(* IEC 61131-3 sources: stc/tests/type_system, 4 files *)

(* ---- init_test.st ---- *)
(* Initialiser test suite (RUNT-06)
   Array, repetition, struct-array, TYPE default and FB-instance
   initialisers apply when the variable is instantiated. Literals are typed
   where the checker's literal adoption would otherwise matter.
*)

TYPE ST_Item :
STRUCT
    id : INT := INT#5;
    name : STRING := 'x';
END_STRUCT
END_TYPE

TYPE T_Speed : INT := INT#50; END_TYPE

FUNCTION_BLOCK FB_Base
VAR
    base_x : INT := INT#3;
END_VAR
END_FUNCTION_BLOCK

FUNCTION_BLOCK FB_Drive EXTENDS FB_Base
VAR_INPUT
    speed : INT;
END_VAR
VAR
    tbl : ARRAY[1..2] OF INT := [INT#4, INT#5];
    item : ST_Item := (name := 'drive');
END_VAR
END_FUNCTION_BLOCK

VAR_GLOBAL CONSTANT
    N_ITEMS : INT := 3;
END_VAR

TEST_CASE 'Array initialiser'
VAR
    arr : ARRAY[1..3] OF INT := [INT#1, INT#2, INT#3];
END_VAR
    ASSERT_EQ(arr[1], INT#1);
    ASSERT_EQ(arr[2], INT#2);
    ASSERT_EQ(arr[3], INT#3);
END_TEST_CASE

TEST_CASE 'Repetition and tail defaults'
VAR
    rep : ARRAY[1..5] OF INT := [3(INT#0), INT#7];
END_VAR
    ASSERT_EQ(rep[3], INT#0);
    ASSERT_EQ(rep[4], INT#7);
    ASSERT_EQ(rep[5], INT#0);
END_TEST_CASE

TEST_CASE 'Struct array over a GVL constant bound'
VAR
    items : ARRAY[1..init_test.N_ITEMS] OF ST_Item := [(id := INT#1, name := 'a'), (id := INT#2)];
END_VAR
    ASSERT_EQ(items[1].name, 'a');
    ASSERT_EQ(items[2].id, INT#2);
    ASSERT_EQ(items[2].name, 'x');
    ASSERT_EQ(items[3].id, INT#5);
END_TEST_CASE

TEST_CASE 'TYPE defaults'
VAR
    s : ST_Item;
    v : T_Speed;
END_VAR
    ASSERT_EQ(s.id, INT#5);
    ASSERT_EQ(v, INT#50);
END_TEST_CASE

TEST_CASE 'FB instances get their own initialised members'
VAR
    d1 : FB_Drive;
    d2 : FB_Drive := (speed := INT#9);
END_VAR
    ASSERT_EQ(d1.base_x, INT#3);
    ASSERT_EQ(d2.tbl[2], INT#5);
    ASSERT_EQ(d2.speed, INT#9);
    d1.item.name := 'changed';
    ASSERT_EQ(d2.item.name, 'drive');
END_TEST_CASE

(* ---- all_types.st ---- *)
(* All Types Declaration File
   Exercises every IEC 61131-3 type supported by the stc toolchain:
   elementary types, arrays, structs, enums, subranges, strings.
*)

(* Enum type declaration *)
TYPE MachineState : (
    MS_IDLE := 0,
    MS_RUNNING := 1,
    MS_FAULT := 2,
    MS_MAINTENANCE := 3
);
END_TYPE

(* Struct type declaration *)
TYPE SensorReading :
STRUCT
    Value     : REAL;
    RawCount  : INT;
    Valid     : BOOL;
    Timestamp : DINT;
    TagName   : STRING;
END_STRUCT;
END_TYPE

(* Subrange type *)
TYPE PercentRange : INT (0..100);
END_TYPE

TYPE MotorSpeed : REAL (0.0..1500.0);
END_TYPE

(* Program using all types *)
PROGRAM TypeShowcase
VAR
    (* Boolean *)
    bFlag : BOOL := TRUE;
    bLatch : BOOL := FALSE;

    (* Integer types *)
    nSint : SINT := -10;
    nInt  : INT := 1000;
    nDint : DINT := 100000;
    nLint : LINT := 1000000;

    (* Unsigned integer types *)
    nUsint : USINT := 200;
    nUint  : UINT := 50000;
    nUdint : UDINT := 4000000;
    nUlint : ULINT := 8000000;

    (* Bit string types *)
    bByte  : BYTE := 16#FF;
    wWord  : WORD := 16#ABCD;
    dwDword : DWORD := 16#12345678;
    lwLword : LWORD := 16#FEDCBA98;

    (* Real types *)
    fReal  : REAL := 3.14;
    fLreal : LREAL := 2.718281828;

    (* String types *)
    sName  : STRING := 'Hello World';
    sEmpty : STRING := '';

    (* Time types *)
    tDelay : TIME := T#500ms;
    tCycle : TIME := T#100ms;

    (* Array *)
    aTemps : ARRAY[1..10] OF REAL;
    aFlags : ARRAY[0..7] OF BOOL;

    (* Enum instance *)
    eState : MachineState := MS_IDLE;

    (* Struct instance *)
    stSensor : SensorReading;

    (* Loop variable *)
    i : INT;
END_VAR
    (* Exercise boolean operators *)
    bLatch := bFlag AND NOT bLatch;
    bLatch := bFlag OR bLatch;
    bLatch := bFlag XOR bLatch;

    (* Exercise integer arithmetic *)
    nInt := nInt + 1;
    nDint := nDint * 2;
    nLint := nLint - 500;

    (* Exercise real arithmetic *)
    fReal := fReal * 2.0;
    fLreal := fLreal + 1.0;

    (* Array operations *)
    FOR i := 1 TO 10 DO
        aTemps[i] := INT_TO_REAL(i) * 10.5;
    END_FOR;

    aFlags[0] := TRUE;
    aFlags[7] := FALSE;

    (* Enum usage *)
    eState := MS_RUNNING;
    IF eState = MS_RUNNING THEN
        nInt := nInt + 100;
    END_IF;

    (* Struct field access *)
    stSensor.Value := 25.4;
    stSensor.RawCount := 1023;
    stSensor.Valid := TRUE;
    stSensor.TagName := 'TT-101';

    (* String operations *)
    sName := CONCAT(sName, '!');
END_PROGRAM

(* ---- type_test.st ---- *)
(* Type System Test Suite
   Validates all elementary types, arithmetic, conversions,
   string operations, arrays, and control flow constructs.
*)

TEST_CASE 'Integer arithmetic on all widths'
VAR
    nSint : SINT := 10;
    nInt  : INT := 1000;
    nDint : DINT := 100000;
    nLint : LINT := 1000000;
END_VAR
    nSint := nSint + 5;
    ASSERT_EQ(nSint, 15);

    nInt := nInt * 2;
    ASSERT_EQ(nInt, 2000);

    nDint := nDint - 50000;
    ASSERT_EQ(nDint, 50000);

    nLint := nLint + 500000;
    ASSERT_EQ(nLint, 1500000);
END_TEST_CASE

TEST_CASE 'Unsigned integer types'
VAR
    nUsint : USINT := 200;
    nUint  : UINT := 50000;
    nUdint : UDINT := 4000000;
END_VAR
    nUsint := nUsint + 55;
    ASSERT_EQ(nUsint, 255);

    nUint := nUint - 10000;
    ASSERT_EQ(nUint, 40000);

    nUdint := nUdint * 2;
    ASSERT_EQ(nUdint, 8000000);
END_TEST_CASE

TEST_CASE 'REAL arithmetic and ASSERT_NEAR'
VAR
    fReal  : REAL := 3.14;
    fLreal : LREAL := 2.718281828;
    result : REAL;
END_VAR
    result := fReal * 2.0;
    ASSERT_NEAR(result, 6.28, 0.001);

    fLreal := fLreal + 1.0;
    ASSERT_NEAR(fLreal, 3.718281828, 0.000001);

    (* Division *)
    result := 10.0 / 3.0;
    ASSERT_NEAR(result, 3.333333, 0.001);
END_TEST_CASE

TEST_CASE 'Boolean logic operators'
VAR
    a : BOOL := TRUE;
    b : BOOL := FALSE;
    r : BOOL;
END_VAR
    r := a AND b;
    ASSERT_FALSE(r);

    r := a OR b;
    ASSERT_TRUE(r);

    r := a XOR b;
    ASSERT_TRUE(r);

    r := NOT a;
    ASSERT_FALSE(r);

    r := a AND NOT b;
    ASSERT_TRUE(r);

    (* Double negation *)
    r := NOT NOT a;
    ASSERT_TRUE(r);
END_TEST_CASE

TEST_CASE 'Comparison operators'
VAR
    x : INT := 10;
    y : INT := 20;
END_VAR
    ASSERT_TRUE(x < y);
    ASSERT_TRUE(y > x);
    ASSERT_TRUE(x <= 10);
    ASSERT_TRUE(y >= 20);
    ASSERT_TRUE(x <> y);
    ASSERT_FALSE(x = y);
    ASSERT_TRUE(x = 10);
END_TEST_CASE

TEST_CASE 'Type conversions INT to REAL'
VAR
    n : INT := 42;
    f : REAL;
END_VAR
    f := INT_TO_REAL(n);
    ASSERT_NEAR(f, 42.0, 0.01);
END_TEST_CASE

TEST_CASE 'Type conversions REAL to INT'
VAR
    f : REAL := 3.7;
    n : INT;
END_VAR
    n := REAL_TO_INT(f);
    ASSERT_EQ(n, 4);  (* Banker's rounding: 3.7 rounds to 4 *)
END_TEST_CASE

TEST_CASE 'Type conversions BOOL to INT and back'
VAR
    b : BOOL := TRUE;
    n : INT;
    b2 : BOOL;
END_VAR
    n := BOOL_TO_INT(b);
    ASSERT_EQ(n, 1);

    b2 := INT_TO_BOOL(0);
    ASSERT_FALSE(b2);

    b2 := INT_TO_BOOL(42);
    ASSERT_TRUE(b2);
END_TEST_CASE

TEST_CASE 'INT to STRING conversion'
VAR
    n : INT := 123;
    s : STRING;
END_VAR
    s := INT_TO_STRING(n);
    ASSERT_EQ(s, '123');
END_TEST_CASE

TEST_CASE 'STRING to INT conversion'
VAR
    s : STRING := '456';
    n : INT;
END_VAR
    n := STRING_TO_INT(s);
    ASSERT_EQ(n, 456);
END_TEST_CASE

TEST_CASE 'String functions: LEN, LEFT, RIGHT, MID'
VAR
    s : STRING := 'Hello World';
    r : STRING;
    n : INT;
END_VAR
    n := LEN(s);
    ASSERT_EQ(n, 11);

    r := LEFT(s, 5);
    ASSERT_EQ(r, 'Hello');

    r := RIGHT(s, 5);
    ASSERT_EQ(r, 'World');

    r := MID(s, 5, 7);  (* 5 chars starting at position 7 *)
    ASSERT_EQ(r, 'World');
END_TEST_CASE

TEST_CASE 'String CONCAT and FIND'
VAR
    s1 : STRING := 'Foo';
    s2 : STRING := 'Bar';
    result : STRING;
    pos : INT;
END_VAR
    result := CONCAT(s1, s2);
    ASSERT_EQ(result, 'FooBar');

    pos := FIND(result, 'Bar');
    ASSERT_EQ(pos, 4);  (* 1-based position *)

    pos := FIND(result, 'xyz');
    ASSERT_EQ(pos, 0);  (* Not found *)
END_TEST_CASE

TEST_CASE 'FOR loop with accumulator'
VAR
    sum : INT := 0;
    i : INT;
END_VAR
    FOR i := 1 TO 10 DO
        sum := sum + i;
    END_FOR;
    ASSERT_EQ(sum, 55);
END_TEST_CASE

TEST_CASE 'FOR loop with BY step'
VAR
    sum : INT := 0;
    i : INT;
END_VAR
    FOR i := 0 TO 10 BY 2 DO
        sum := sum + i;
    END_FOR;
    (* 0+2+4+6+8+10 = 30 *)
    ASSERT_EQ(sum, 30);
END_TEST_CASE

TEST_CASE 'WHILE loop'
VAR
    count : INT := 0;
    value : INT := 1;
END_VAR
    WHILE value < 100 DO
        value := value * 2;
        count := count + 1;
    END_WHILE;
    (* 1->2->4->8->16->32->64->128, 7 iterations *)
    ASSERT_EQ(count, 7);
    ASSERT_EQ(value, 128);
END_TEST_CASE

TEST_CASE 'REPEAT-UNTIL loop'
VAR
    n : INT := 10;
    count : INT := 0;
END_VAR
    REPEAT
        n := n - 3;
        count := count + 1;
    UNTIL n <= 0
    END_REPEAT;
    (* 10->7->4->1->-2: 4 iterations *)
    ASSERT_EQ(count, 4);
    ASSERT_TRUE(n <= 0);
END_TEST_CASE

TEST_CASE 'CASE statement with integer labels'
VAR
    cmd : INT := 2;
    result : STRING := '';
END_VAR
    CASE cmd OF
        0: result := 'STOP';
        1: result := 'SLOW';
        2: result := 'RUN';
        3: result := 'FAST';
    ELSE
        result := 'UNKNOWN';
    END_CASE;
    ASSERT_EQ(result, 'RUN');
END_TEST_CASE

TEST_CASE 'CASE statement ELSE branch'
VAR
    cmd : INT := 99;
    result : STRING := '';
END_VAR
    CASE cmd OF
        0: result := 'STOP';
        1: result := 'RUN';
    ELSE
        result := 'UNKNOWN';
    END_CASE;
    ASSERT_EQ(result, 'UNKNOWN');
END_TEST_CASE

TEST_CASE 'Nested IF-ELSIF-ELSE'
VAR
    temp : REAL := 85.0;
    alarm : INT := 0;
END_VAR
    IF temp > 100.0 THEN
        alarm := 3;  (* Critical *)
    ELSIF temp > 80.0 THEN
        alarm := 2;  (* Warning *)
    ELSIF temp > 60.0 THEN
        alarm := 1;  (* Advisory *)
    ELSE
        alarm := 0;  (* Normal *)
    END_IF;
    ASSERT_EQ(alarm, 2);
END_TEST_CASE

TEST_CASE 'EXIT breaks out of loop'
VAR
    i : INT;
    last : INT := 0;
END_VAR
    FOR i := 1 TO 100 DO
        IF i > 5 THEN
            EXIT;
        END_IF;
        last := i;
    END_FOR;
    ASSERT_EQ(last, 5);
END_TEST_CASE

TEST_CASE 'Negative integer arithmetic'
VAR
    a : INT := -10;
    b : INT := 3;
    r : INT;
END_VAR
    r := a + b;
    ASSERT_EQ(r, -7);

    r := a * b;
    ASSERT_EQ(r, -30);

    r := a - b;
    ASSERT_EQ(r, -13);
END_TEST_CASE

TEST_CASE 'REAL precision with small values'
VAR
    a : REAL := 0.1;
    b : REAL := 0.2;
    sum : REAL;
END_VAR
    sum := a + b;
    (* Floating point: 0.1+0.2 is not exactly 0.3 *)
    ASSERT_NEAR(sum, 0.3, 0.001);
END_TEST_CASE

TEST_CASE 'Multiple assignments in sequence'
VAR
    x : INT;
    y : INT;
    z : INT;
END_VAR
    x := 1;
    y := x + 1;
    z := y + 1;
    ASSERT_EQ(x, 1);
    ASSERT_EQ(y, 2);
    ASSERT_EQ(z, 3);
END_TEST_CASE

(* ---- wrap_test.st ---- *)
(* Integer wrap-around test suite (RUNT-05)
   Typed integer stores and typed arithmetic wrap to the IEC width of the
   type. Operands use typed literals so the suite does not depend on the
   checker adopting untyped literals.
*)

TEST_CASE 'INT wraps from 32767 to -32768'
VAR
    i : INT := INT#32767;
END_VAR
    i := i + INT#1;
    ASSERT_EQ(i, INT#-32768);
    i := i - INT#1;
    ASSERT_EQ(i, INT#32767);
END_TEST_CASE

TEST_CASE 'UINT wraps from 0 to 65535'
VAR
    u : UINT;
END_VAR
    u := u - UINT#1;
    ASSERT_EQ(u, UINT#65535);
    u := u + UINT#1;
    ASSERT_EQ(u, UINT#0);
END_TEST_CASE

TEST_CASE 'Byte-wide types wrap'
VAR
    b : BYTE := BYTE#255;
    s : SINT := SINT#127;
    us : USINT;
END_VAR
    b := b + BYTE#1;
    ASSERT_EQ(b, BYTE#0);
    s := s + SINT#1;
    ASSERT_EQ(s, SINT#-128);
    us := us - USINT#1;
    ASSERT_EQ(us, USINT#255);
END_TEST_CASE

TEST_CASE 'DINT and UDINT wrap'
VAR
    d : DINT := DINT#2147483647;
    ud : UDINT;
END_VAR
    d := d + DINT#1;
    ASSERT_EQ(d, DINT#-2147483648);
    ud := ud - UDINT#1;
    ASSERT_EQ(ud, UDINT#4294967295);
END_TEST_CASE
